(* IEC 61131-3 sources: ZUT-informatyka/Semestr 5/PUA, 3 files *)

(* ---- Types.typ ---- *)
TYPE
	RoomStruct : STRUCT
		diToogle : ARRAY[1..2] OF BOOL; (* Wlaczniki *)
		doLamp : ARRAY[1..2] OF BOOL; (* Lampy *)
		aiTemperature : INT; (* Temperatura *)
		diPhotoCom : ARRAY[1..2] OF BOOL; (* Fotokomorka *)
		aiDimmer : ARRAY[1..2] OF INT; (* Obsluga sciemniacza *)
		aoLamp : ARRAY[1..2] OF INT; (* Obsluga lampy sciemnianej *)
		Dryer : DryerStruct;
	END_STRUCT;

	StairsStruct : STRUCT
		diParter : BOOL;
		diPietro : BOOL;
		doLamp : BOOL;
	END_STRUCT;

	HouseStruct : STRUCT
		Jadalnia : RoomStruct;
		Kuchnia : RoomStruct;
		Sypialnia : RoomStruct;
		Korytarz : RoomStruct;
		Schody : StairsStruct;
		Lazienka : RoomStruct;
	END_STRUCT;

	OperatorStruct : STRUCT
		diStart : BOOL;
		diStop : BOOL;
		diEStop : BOOL;
		doAktywny : BOOL;
		doAwaria : BOOL;
		diReset : BOOL;
		aiSetter : INT;
	END_STRUCT;

	EngineStruct : STRUCT
		diTermikNO : BOOL; (* Czujnik termiczny : TRUE - za wysoka temperatura, FALSE - temperatura OK => DI11 *)
		diTermikNC : BOOL; (* Czujnik termiczny : FALSE - za wysoka temperatura, TRUE - temperatura OK => DI12 *)
		doOnOff : BOOL; (* Wysterowanie silnika *)
	END_STRUCT;

	SensorNONCStruct : STRUCT
		uiSetValue : INT;
		uiOutNC : BOOL;
		uiOutNO : BOOL;
	END_STRUCT;

	TankStruct : STRUCT
		doHeater : BOOL; (* Odpowiednik pompy w hydroforze *)
		diTermik : BOOL; (* Odpowiednik zabezpieczenia stykow silnika pompy w hydroforze *)
		aiTemperature : INT;
		aoHeater : INT;
		aoFan : INT;
		uiHeaterSetValue : INT;
		ThermoMin : SensorNONCStruct;
		ThermoMax : SensorNONCStruct;
	END_STRUCT;

	StatisticsStruct : STRUCT
		uiWorkTime : ARRAY[1..10] OF TimeStruct;
	END_STRUCT;

	TimeStruct : STRUCT
		uiSeconds : USINT;
		uiMinues : USINT;
		uiHours : DINT;
	END_STRUCT;

	DryerStruct : STRUCT
		diHand : BOOL; (* czujnik wykrywania rak - laser lub fotokomroka NO/NC *)
		diTermik : BOOL; (* czujnik przeciazeniowy stycznika zalaczajacego grzalke i wentylator NO/NC *)
		doDryer : BOOL; (* stycznik -> wentylator i grzalka *)
	END_STRUCT;

	StateMachineEnum : (
		INIT := 1,
		HEAT_UP := 2,
		TEMP_CONST := 3,
		HEAT_DOWN := 4,
		WAIT_STOP := 5,
		FAILURE := 6,
		STOP_TEMP := 7
	);

	FurnaceStruct : STRUCT
		aoHeater : INT;
		aoFan : INT;
		aiTemperature : INT;
		uiHeater : REAL;
		uiFan : REAL;
		uiTemperature : REAL;
		diTempFailure : BOOL;
		uiTempFailure : BOOL;
	END_STRUCT;

	HeatingSystemStruct : STRUCT
		Operator : OperatorStruct;
		Furnace : FurnaceStruct;
	END_STRUCT;

	HeatingSystemParStruct : STRUCT
		uiSetTime : ARRAY[1..10] OF REAL;
		uiSetTemperature : ARRAY[1..10] OF REAL;
	END_STRUCT;
END_TYPE

(* ---- Main.st ---- *)
PROGRAM _INIT
	(* Insert code here *)
	uiLightControl := 9;
	//uiClockTON_PT[1] := 1;
	Tank.uiHeaterSetValue := 15000;
	Tank.ThermoMin.uiSetValue := 550;
	Tank.ThermoMax.uiSetValue := 600;
	uiCycleTime := 10;
	StateMachine := INIT;

	HeatingSystemPar.uiSetTime[1] := 120;
	HeatingSystemPar.uiSetTime[2] := 15;
END_PROGRAM

PROGRAM _CYCLIC
	(* Insert code here *)
	CASE uiLightControl OF
		1 : // Klasyczne sterowanie
			Home.Jadalnia.doLamp[1] := Home.Jadalnia.diToogle[1];

		2: // Dotyk
			Home.Jadalnia.doLamp[1] := EDGEPOS(Home.Jadalnia.diToogle[1]) XOR Home.Jadalnia.doLamp[1];

		3: // Mrugajace
			ClockTON[1].IN := Home.Jadalnia.diToogle[2] AND NOT (ClockTON[1].Q);
			//ClockTON[1].PT := REAL_TO_TIME(uiClockTON_PT[1] * 1000);
			ClockTON[1]();
			Home.Jadalnia.doLamp[1] := Home.Jadalnia.diToogle[2] AND (ClockTON[1].Q XOR Home.Jadalnia.doLamp[1]);

			IF EDGEPOS(Home.Jadalnia.doLamp[1]) THEN
				ClockTON[1].PT := REAL_TO_TIME(uiClockTON_PT[1] * 1000);
			END_IF;
			IF EDGENEG(Home.Jadalnia.doLamp[1]) THEN
				ClockTON[1].PT := REAL_TO_TIME(uiClockTON_PT[2] * 1000);
			END_IF;

		4: // Fotokomorka
			ClockTOF[1].IN := Home.Korytarz.diPhotoCom[1];
			ClockTOF[1].PT := REAL_TO_TIME(uiClockTOF_PT[1] * 1000);
			ClockTOF[1]();
			Home.Korytarz.doLamp[1] := ClockTOF[1].Q;

		5: // Potencjometr
			(*
			Scale[1].x := INT_TO_REAL(Home.Jadalnia.aiDimmer[1]); // Obsluga potencjometrem
			Scale[1].x1 := 4;
			Scale[1].y1 := 14000;
			Scale[1].x2 := 32767;
			Scale[1].y2 := 28000;
			Scale[1]();
			Home.Jadalnia.aoLamp[1] := REAL_TO_INT(Scale[1].y);
			*)
			Scale[2].x := INT_TO_REAL(Home.Jadalnia.aiDimmer[2]); // Obsluga termometrem
			Scale[2].x1 := 290;
			Scale[2].y1 := 14000;
			Scale[2].x2 := 350;
			Scale[2].y2 := 28000;
			Scale[2]();
			Home.Jadalnia.aoLamp[1] := REAL_TO_INT(Scale[2].y);

		6: // Schodowy
			//Home.Schody.doLamp := Home.Schody.diParter AND NOT (Home.Schody.diPietro) OR NOT (Home.Schody.diParter) AND Home.Schody.diPietro;
			Home.Schody.doLamp := Home.Schody.diParter XOR Home.Schody.diPietro;
			IF Home.Schody.doLamp THEN
				Home.Jadalnia.aoLamp[1] := 20000;
			ELSE
				Home.Jadalnia.aoLamp[1] := 0;
			END_IF

		7: // Procedura start stop
			//Operator.doAktywny := (EDGEPOS(Operator.diStart) OR Operator.doAktywny) AND NOT (Operator.diStop) AND NOT(Operator.doAwaria); (* Start odpali sie tylko raz *)
			//Operator.doAwaria := Engine.diTermikNC OR (Operator.doAwaria AND NOT(Operator.diReset));

			Operator.doAwaria := Engine.diTermikNC OR (Operator.doAwaria AND NOT(Operator.diReset));

			fRS[1].SET := EDGEPOS(Operator.diStart);
			fRS[1].RESET1 := Operator.diStop OR Operator.doAwaria (* OR Operator.diEStop *);
			fRS[1]();
			Operator.doAktywny := fRS[1].Q1;

			fSR[1].SET1 := Tank.diTermik OR Operator.diEStop;
			fSR[1].RESET := Operator.diReset;
			fSR[1]();
			Operator.doAwaria := fSR[1].Q1;

			// Obsluga termostatu
			IF Tank.aiTemperature >= Tank.ThermoMax.uiSetValue THEN // Poziom temperatury wylaczania
				Tank.ThermoMax.uiOutNC := FALSE;
				Tank.ThermoMax.uiOutNO := TRUE;
			ELSE
				Tank.ThermoMax.uiOutNC := TRUE;
				Tank.ThermoMax.uiOutNO := FALSE;
			END_IF;

			IF Tank.aiTemperature >= Tank.ThermoMin.uiSetValue THEN // Poziom temperatury wlaczania
				Tank.ThermoMin.uiOutNC := FALSE;
				Tank.ThermoMin.uiOutNO := TRUE;
			ELSE
				Tank.ThermoMin.uiOutNC := TRUE;
				Tank.ThermoMin.uiOutNO := FALSE;
			END_IF;

			IF Tank.doHeater THEN // Obsluga grzalki
				Tank.aoHeater := Tank.uiHeaterSetValue;
			ELSE
				Tank.aoHeater := 0;
			END_IF;

			fRS[2].SET := Tank.ThermoMin.uiOutNC AND Operator.doAktywny;
			fRS[2].RESET1 := NOT(Tank.ThermoMax.uiOutNC) OR Operator.diStop;
			fRS[2]();
			Tank.doHeater := fRS[2].Q1;
			Tank.aoFan := Operator.aiSetter; // Obsluga wentylatora

			// Pomiar czasu pracy
			ClockTON[2].IN := Tank.doHeater AND NOT(ClockTON[2].Q);
			ClockTON[2].PT := T#1s;
			ClockTON[2]();

			IF ClockTON[2].Q THEN
	  			Statistic.uiWorkTime[1].uiSeconds := Statistic.uiWorkTime[1].uiSeconds + 1;
			END_IF;
			IF Statistic.uiWorkTime[1].uiSeconds >= 60 THEN
				Statistic.uiWorkTime[1].uiSeconds := 0;
				Statistic.uiWorkTime[1].uiMinues := Statistic.uiWorkTime[1].uiMinues + 1;
			END_IF;
			IF Statistic.uiWorkTime[1].uiMinues >= 60 THEN
				Statistic.uiWorkTime[1].uiMinues := 0;
				Statistic.uiWorkTime[1].uiHours := Statistic.uiWorkTime[1].uiHours + 1;
			END_IF;
			IF EDGEPOS(Operator.doAktywny) THEN
				Statistic.uiWorkTime[1].uiSeconds := 0;
				Statistic.uiWorkTime[1].uiMinues := 0;
				Statistic.uiWorkTime[1].uiHours := 0;
			END_IF;

		8: // obsluga suszarki do rak + pomiary czasu
			ClockTOF[3].IN := Home.Lazienka.Dryer.diHand;
			ClockTOF[3].PT := T#0.5s;
			ClockTOF[3]();
			ClockTON[3].IN := ClockTOF[3].Q;
			ClockTON[3].PT := T#15s;
			ClockTON[3]();
			Home.Lazienka.Dryer.doDryer := NOT(ClockTON[3].Q) AND ClockTOF[3].Q;

			// Pomiar czasu pracy
			ClockTON[2].IN := Home.Lazienka.Dryer.doDryer AND NOT(ClockTON[2].Q);
			ClockTON[2].PT := T#1s;
			ClockTON[2]();

			IF ClockTON[2].Q THEN
				Statistic.uiWorkTime[3].uiSeconds := Statistic.uiWorkTime[3].uiSeconds + 1;
			END_IF;
			IF Statistic.uiWorkTime[3].uiSeconds >= 60 THEN
				Statistic.uiWorkTime[3].uiSeconds := 0;
				Statistic.uiWorkTime[3].uiMinues := Statistic.uiWorkTime[3].uiMinues + 1;
			END_IF;
			IF Statistic.uiWorkTime[3].uiMinues >= 60 THEN
				Statistic.uiWorkTime[3].uiMinues := 0;
				Statistic.uiWorkTime[3].uiHours := Statistic.uiWorkTime[3].uiHours + 1;
			END_IF;
			IF EDGEPOS(Operator.diReset) THEN
				Statistic.uiWorkTime[3].uiSeconds := 0;
				Statistic.uiWorkTime[3].uiMinues := 0;
				Statistic.uiWorkTime[3].uiHours := 0;
			END_IF;

			IF EDGEPOS((TIME_TO_DINT(ClockTON[3].ET) MOD 1000) = 0) AND (TIME_TO_DINT(ClockTON[3].ET) > 0) THEN
				Statistic.uiWorkTime[4].uiSeconds := Statistic.uiWorkTime[4].uiSeconds + 1;
			END_IF;
			IF Statistic.uiWorkTime[4].uiSeconds >= 60 THEN
				Statistic.uiWorkTime[4].uiSeconds := 0;
				Statistic.uiWorkTime[4].uiMinues := Statistic.uiWorkTime[4].uiMinues + 1;
			END_IF;
			IF Statistic.uiWorkTime[4].uiMinues >= 60 THEN
				Statistic.uiWorkTime[4].uiMinues := 0;
				Statistic.uiWorkTime[4].uiHours := Statistic.uiWorkTime[4].uiHours + 1;
			END_IF;
			IF EDGEPOS(Operator.diReset) THEN
				Statistic.uiWorkTime[4].uiSeconds := 0;
				Statistic.uiWorkTime[4].uiMinues := 0;
				Statistic.uiWorkTime[4].uiHours := 0;
			END_IF;

			IF Home.Lazienka.Dryer.doDryer THEN
				i := i + 1;
			END_IF;

			// zegar polegajacy na czasie cyklu
			IF i >= uiCycleTime THEN
				Statistic.uiWorkTime[5].uiSeconds := Statistic.uiWorkTime[5].uiSeconds + 1;
				i := 0;
			END_IF;
			IF Statistic.uiWorkTime[5].uiSeconds >= 60 THEN
				Statistic.uiWorkTime[5].uiSeconds := 0;
				Statistic.uiWorkTime[5].uiMinues := Statistic.uiWorkTime[5].uiMinues + 1;
			END_IF;
			IF Statistic.uiWorkTime[5].uiMinues >= 60 THEN
				Statistic.uiWorkTime[5].uiMinues := 0;
				Statistic.uiWorkTime[5].uiHours := Statistic.uiWorkTime[5].uiHours + 1;
			END_IF;
			IF EDGEPOS(Operator.diReset) THEN
				Statistic.uiWorkTime[5].uiSeconds := 0;
				Statistic.uiWorkTime[5].uiMinues := 0;
				Statistic.uiWorkTime[5].uiHours := 0;
			END_IF;

		9: // synteza maszyny stanow dla piecyka
			CASE StepNumber OF
				2..4:
					IF cOnOff.error >= cOnOffPar.E_max THEN
						cOnOff.outCV := cOnOffPar.CV_max; // grzej
					END_IF
					IF cOnOff.error <= cOnOffPar.E_min THEN
						cOnOff.outCV := cOnOffPar.CV_min; // nie grzej
					END_IF

				1,5..7:
					cOnOff.outCV := 0;
			END_CASE;

			HeatingSystem.Furnace.uiTemperature := INT_TO_REAL(HeatingSystem.Furnace.aiTemperature);
			cOnOff.error := HeatingSystemPar.uiSetTemperature[1] - HeatingSystem.Furnace.aiTemperature;

			HeatingSystem.Furnace.aoHeater := REAL_TO_INT(cOnOff.outCV);
			HeatingSystem.Furnace.aoFan := HeatingSystem.Operator.aiSetter;

			CASE StateMachine OF
				INIT:
					StepNumber := 1;
					fRS[1].SET := HeatingSystem.Operator.diStart;
					fRS[1].RESET1 := HeatingSystem.Operator.diStop;
					fRS[1]();
					HeatingSystem.Operator.doAktywny := fRS[1].Q1;

					IF HeatingSystem.Operator.doAktywny THEN
						HeatingSystemPar.uiSetTemperature[1] := 500;
						StateMachine := HEAT_UP;
					END_IF

				HEAT_UP:
					StepNumber := 2;
					IF EDGEPOS(HeatingSystem.Operator.diStop) THEN
						StateMachine := STOP_TEMP;
					END_IF
					IF HeatingSystem.Furnace.uiTemperature >= HeatingSystemPar.uiSetTemperature[1] THEN
						StateMachine := TEMP_CONST;
					END_IF

				TEMP_CONST:
					StepNumber := 3;
					ClockTON[5].IN := TRUE;
					ClockTON[5].PT := REAL_TO_TIME(HeatingSystemPar.uiSetTime[1] * 1000);
					ClockTON[5]();
					IF EDGEPOS(HeatingSystem.Operator.diStop) THEN
						StateMachine := STOP_TEMP;
					END_IF
					IF ClockTON[5].Q THEN
						ClockTON[5].IN := FALSE;
						ClockTON[5]();
						HeatingSystemPar.uiSetTemperature[1] := 400;
						StateMachine := HEAT_DOWN;
					END_IF

				HEAT_DOWN:
					StepNumber := 4;
					IF EDGEPOS(HeatingSystem.Operator.diStop) THEN
						StateMachine := STOP_TEMP;
					END_IF
					IF HeatingSystem.Furnace.uiTemperature <= HeatingSystemPar.uiSetTemperature[1] THEN
						StateMachine := WAIT_STOP;
					END_IF

				WAIT_STOP:
					StepNumber := 5;
					ClockTON[5].IN := TRUE;
					ClockTON[5].PT := REAL_TO_TIME(HeatingSystemPar.uiSetTime[2] * 1000);
					ClockTON[5]();
					IF ClockTON[5].Q THEN
						ClockTON[5].IN := FALSE;
						ClockTON[5]();
						//HeatingSystem.Operator.doAktywny := FALSE;
						StateMachine := INIT;
					END_IF
					IF EDGEPOS(HeatingSystem.Operator.diStop) THEN
						StateMachine := STOP_TEMP;
					END_IF

				FAILURE:
					StepNumber := 6;
					IF EDGEPOS(HeatingSystem.Operator.diStop) THEN
						HeatingSystem.Operator.doAktywny := FALSE; // dezaktywacja systemu
						StateMachine := INIT;
					END_IF

				STOP_TEMP:
					StepNumber := 7;
					IF EDGEPOS(HeatingSystem.Operator.diStop) THEN
						HeatingSystem.Operator.doAktywny := FALSE; // dezaktywacja systemu
						StateMachine := INIT;
					END_IF
			END_CASE;
	END_CASE;
END_PROGRAM

PROGRAM _EXIT
	(* Insert code here *)

END_PROGRAM

(* ---- Variables.var ---- *)
VAR
	Home : HouseStruct;
	uiLightControl : USINT; (* Tryby pracy oswietlenia 1 : klasyczne sterowanie, 2 : dotyk, 3 : swiatlo pulsujace ze stalym zboczem, 4 : swiatlo pulsujace ze zmiennym zboczem*)
	ClockTON : ARRAY[1..10] OF TON;
	ClockTOF : ARRAY[1..10] OF TOF;
	Scale : ARRAY[1..10] OF LCRLimScal;
	Operator : OperatorStruct;
	Engine : EngineStruct;
	fSR : ARRAY[1..10] OF SR;
	fRS : ARRAY[1..10] OF RS;
	Tank : TankStruct;
	i : USINT;
	uiCycleTime : USINT;
	StepNumber : USINT;
	HeatingSystem : HeatingSystemStruct;
	StateMachine : StateMachineEnum;
	cOnOff : cOnOffStruct;
END_VAR

VAR RETAIN
	uiClockTON_PT : ARRAY[1..10] OF REAL; (* Czas zadany w sekundach *)
	uiClockTOF_PT : ARRAY[1..10] OF REAL; (* Czas zadany w sekundach *)
	Statistic : StatisticsStruct;
	HeatingSystemPar : HeatingSystemParStruct;
	cOnOffPar : cOnOffParStruct;
END_VAR
